// TIA Portal V18 export
TYPE "DI16x24V_In"
   STRUCT
      Ch0 : Bool;
      Ch1 : Bool;
      Ch2 : Bool;
      Ch3 : Bool;
      Ch4 : Bool;
      Ch5 : Bool;
      Ch6 : Bool;
      Ch7 : Bool;
      Ch8 : Bool;
      Ch9 : Bool;
      Ch10 : Bool;
      Ch11 : Bool;
      Ch12 : Bool;
      Ch13 : Bool;
      Ch14 : Bool;
      Ch15 : Bool;
   END_STRUCT;
END_TYPE
